FUNCTION_BLOCK vaccum3 (* Basic Function Block Type *)
  (* Standard: 61499-2 *)
  (* Version 0.0, 2011-02-26, Majid Sorouri, nxtControl GmbH, Template *)
  (* Compiler header: package fb.rt.pnp; *)
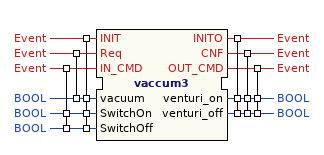
  EVENT_INPUT
    INIT WITH vacuum, SwitchOn, SwitchOff; (* Initialization Request *)
    Req WITH vacuum;
    IN_CMD WITH SwitchOn, SwitchOff;
  END_EVENT
  EVENT_OUTPUT
    INITO WITH venturi_on, venturi_off; (* Initialization Confirm *)
    CNF WITH venturi_on, venturi_off;
    OUT_CMD WITH venturi_on, venturi_off; (* Execution Confirmation *)
  END_EVENT
  VAR_INPUT
    vacuum : BOOL;
    SwitchOn : BOOL;
    SwitchOff : BOOL;
  END_VAR
  VAR_OUTPUT
    venturi_on : BOOL; (* Output event qualifier *)
    venturi_off : BOOL;
  END_VAR
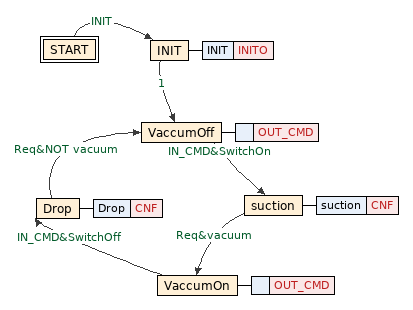
  EC_STATES
    START; (* Initial State *)
    INIT : INIT -> INITO; (* Initialization *)
    suction : suction -> CNF;
    Drop : Drop -> CNF;
    VaccumOn : -> OUT_CMD;
    VaccumOff : -> OUT_CMD;
  END_STATES
  EC_TRANSITIONS
    START TO INIT := INIT;
    INIT TO VaccumOff := 1;
    VaccumOff TO suction := IN_CMD&SwitchOn;
    VaccumOn TO Drop := IN_CMD&SwitchOff;
    Drop TO VaccumOff := Req&NOT vacuum;
    suction TO VaccumOn := Req&vacuum;
  END_TRANSITIONS
  ALGORITHM INIT IN ST: (* Initialization algorithm *)
venturi_off:=TRUE;
venturi_on:=FALSE;
System.out.println("Vassum3 INIT");
  END_ALGORITHM
  ALGORITHM suction IN ST:
venturi_off:=FALSE;
venturi_on:=TRUE;
System.out.println("Vaccum3 Suction");
  END_ALGORITHM
  ALGORITHM Drop IN ST:
venturi_off:=TRUE;
venturi_on:=FALSE;
System.out.println("Vaccum3 Drop");
  END_ALGORITHM
END_FUNCTION_BLOCK
